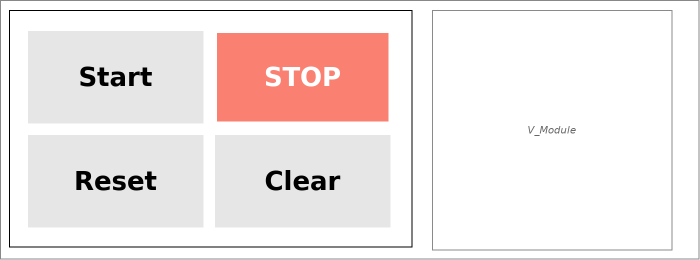
VISUALIZATION V_MachineModule  // 700x260
VAR_IN_OUT
	HMI : ST_PackMLBaseModule_HMI;
END_VAR
    Frame (432,10 240x240)
        shows V_Module(HMI := HMI)
    RoundedRectangle (9,10 403x237)
    RoundedRectangle (28,31 175x92), "Start"
        OnMouseClick: execute { HMI.Command.State := E_PMLCommand.ePMLCommand_Start; }
    RoundedRectangle (215,135 175x92), "Clear"
        OnMouseClick: execute { HMI.Command.State := E_PMLCommand.ePMLCommand_Clear; }
    RoundedRectangle (28,135 175x92), "Reset"
        OnMouseClick: execute { HMI.Command.State := E_PMLCommand.ePMLCommand_Reset; }
    RoundedRectangle (215,31 175x92), "STOP"
        toggle SafetyGlobalVariableList.eStopHMI
        OnMouseClick: execute { HMI.Command.State := E_PMLCommand.ePMLCommand_Clear; }
END_VISUALIZATION

(* stored: Version 1.1.0.1, ProductVersion 3.1.4024.12
   Visu V_MachineModule: Id {52e6719a-8063-4140-8dd7-11f9fb20ffd0} *)
